% RSLogix 500 project project1.RSS, saved by version 8.30.00.16 %
PROJECT "UNTITLED"    % processor: Bul.1763 MicroLogix 1100 Series A %

PROGRAM FILES
  LAD 2 "MAIN"  4 rungs
  LAD 3 "INPUTS"  3 rungs
  LAD 4 "OUTPUTS"  3 rungs
  LAD 5 "CONTROLS"  11 rungs

DATA FILES
  O0 OUTPUT  5 elements
  I1 INPUT  7 elements
  S2 STATUS  66 elements
  B3 BINARY  3 elements
  T4 TIMER  4 elements
  C5 COUNTER  1 elements
  R6 CONTROL  1 elements
  N7 INTEGER  1 elements
  F8 FLOAT  1 elements

LADDER 2 "MAIN"
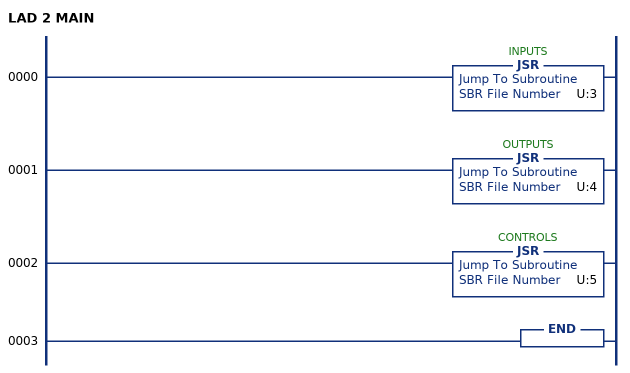
% Rung: 0 %
SOR JSR U:3 EOR
%   U:3  "INPUTS" %
% Rung: 1 %
SOR JSR U:4 EOR
%   U:4  "OUTPUTS" %
% Rung: 2 %
SOR JSR U:5 EOR
%   U:5  "CONTROLS" %
% Rung: 3 %
SOR END EOR

LADDER 3 "INPUTS"
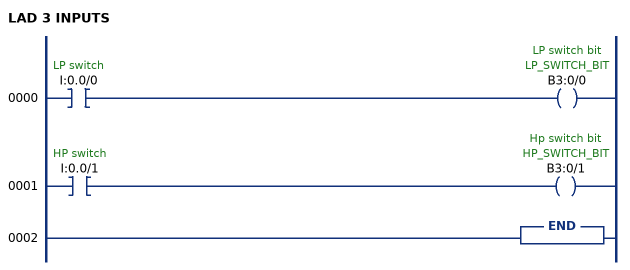
% Rung: 0 %
SOR XIC I:0.0/0 OTE B3:0/0 EOR
%   I:0.0/0  "LP switch" %
%   B3:0/0  LP_SWITCH_BIT  "LP switch bit" %
% Rung: 1 %
SOR XIC I:0.0/1 OTE B3:0/1 EOR
%   I:0.0/1  "HP switch" %
%   B3:0/1  HP_SWITCH_BIT  "Hp switch bit" %
% Rung: 2 %
SOR END EOR

LADDER 4 "OUTPUTS"
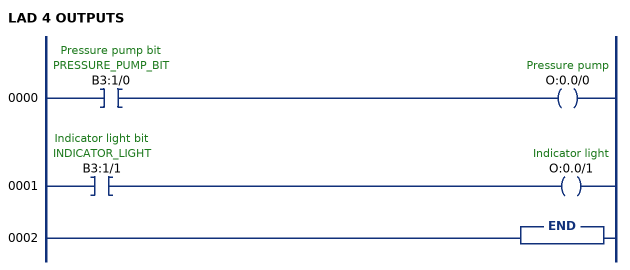
% Rung: 0 %
SOR XIC B3:1/0 OTE O:0.0/0 EOR
%   B3:1/0  PRESSURE_PUMP_BIT  "Pressure pump bit" %
%   O:0.0/0  "Pressure pump" %
% Rung: 1 %
SOR XIC B3:1/1 OTE O:0.0/1 EOR
%   B3:1/1  INDICATOR_LIGHT  "Indicator light bit" %
%   O:0.0/1  "Indicator light" %
% Rung: 2 %
SOR END EOR

LADDER 5 "CONTROLS"
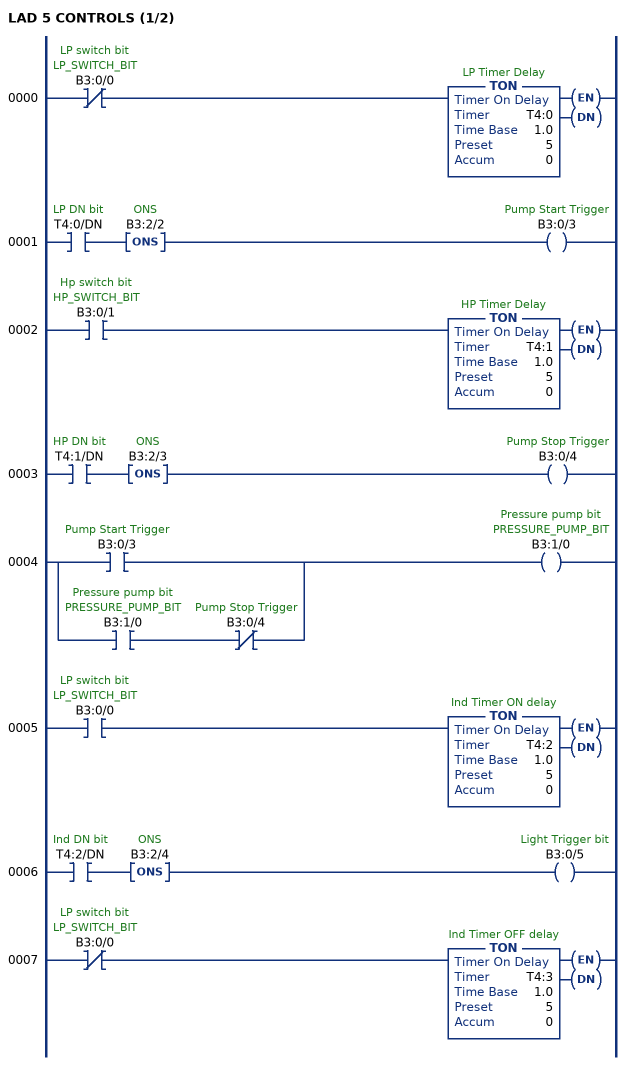
% Rung: 0 %
SOR XIO B3:0/0 TON T4:0 1.0 5 0 EOR
%   B3:0/0  LP_SWITCH_BIT  "LP switch bit" %
%   T4:0  "LP Timer Delay" %
% Rung: 1 %
SOR XIC T4:0/DN ONS B3:2/2 OTE B3:0/3 EOR
%   T4:0/DN  "LP DN bit" %
%   B3:2/2  "ONS" %
%   B3:0/3  "Pump Start Trigger" %
% Rung: 2 %
SOR XIC B3:0/1 TON T4:1 1.0 5 0 EOR
%   B3:0/1  HP_SWITCH_BIT  "Hp switch bit" %
%   T4:1  "HP Timer Delay" %
% Rung: 3 %
SOR XIC T4:1/DN ONS B3:2/3 OTE B3:0/4 EOR
%   T4:1/DN  "HP DN bit" %
%   B3:2/3  "ONS" %
%   B3:0/4  "Pump Stop Trigger" %
% Rung: 4 %
SOR BST XIC B3:0/3 NXB XIC B3:1/0 XIO B3:0/4 BND OTE B3:1/0 EOR
%   B3:0/3  "Pump Start Trigger" %
%   B3:1/0  PRESSURE_PUMP_BIT  "Pressure pump bit" %
%   B3:0/4  "Pump Stop Trigger" %
% Rung: 5 %
SOR XIC B3:0/0 TON T4:2 1.0 5 0 EOR
%   B3:0/0  LP_SWITCH_BIT  "LP switch bit" %
%   T4:2  "Ind Timer ON delay" %
% Rung: 6 %
SOR XIC T4:2/DN ONS B3:2/4 OTE B3:0/5 EOR
%   T4:2/DN  "Ind DN bit" %
%   B3:2/4  "ONS" %
%   B3:0/5  "Light Trigger bit" %
% Rung: 7 %
SOR XIO B3:0/0 TON T4:3 1.0 5 0 EOR
%   B3:0/0  LP_SWITCH_BIT  "LP switch bit" %
%   T4:3  "Ind Timer OFF delay" %

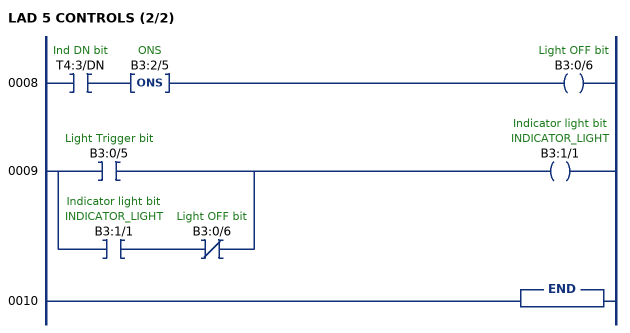
% Rung: 8 %
SOR XIC T4:3/DN ONS B3:2/5 OTE B3:0/6 EOR
%   T4:3/DN  "Ind DN bit" %
%   B3:2/5  "ONS" %
%   B3:0/6  "Light OFF bit" %
% Rung: 9 %
SOR BST XIC B3:0/5 NXB XIC B3:1/1 XIO B3:0/6 BND OTE B3:1/1 EOR
%   B3:0/5  "Light Trigger bit" %
%   B3:1/1  INDICATOR_LIGHT  "Indicator light bit" %
%   B3:0/6  "Light OFF bit" %
% Rung: 10 %
SOR END EOR

OTHER DOCUMENTED ADDRESSES
  B3:0/2  "LP DN bit"
  B3:2/0  SYSTEM_MODE  "System mode"
  B3:2/1  "system mode 1"

DATA TABLE (non-zero values as saved)
DATA T4
% .PRE .ACC %
% T4:0 % 5 0
% T4:1 % 5 0
% T4:2 % 5 0
% T4:3 % 5 0
